TEXTLIST Leak_Detection_Fault
  0 = 'HEALTHY'
  1 = 'FAULT'
   = ''
END_TEXTLIST

(* stored: Version 1.1.0.1, ProductVersion 3.1.4024.12
   TextList Leak_Detection_Fault: Id {8bf4f302-d2bf-4211-bf7b-58cc46bff588} *)
